(* PLC project Untitled1, Eclipse Foundation CIF to Structured Text 0.0 *)
(* stored: creationDateTime 1970-01-01T00:00:00Z *)

TYPE STATE : STRUCT
  curTime : LREAL;
  dvar_M_aut_i AT %Q* : DINT;
  dvar_M_aut_j AT %Q* : DINT;
  dvar_M_aut_l AT %Q* : ARRAY[0..4] OF DINT;
  dvar_M_aut_ll AT %Q* : ARRAY[0..1] OF ARRAY[0..4] OF DINT;
  dvar_M_aut_empty_arr AT %Q* : ARRAY[0..0] OF DINT;
  dvar_M_aut AT %Q* : enum_E;
END_STRUCT;
END_TYPE

TYPE enum_E : (elit_l1, elit_l2, elit_l3, elit_l4, elit_l5, elit_l6, elit_l7, elit_l8);
END_TYPE

FUNCTION makeArray0 : ARRAY[0..4] OF DINT
  VAR_INPUT
    elem0 : DINT;
    elem1 : DINT;
    elem2 : DINT;
    elem3 : DINT;
    elem4 : DINT;
  END_VAR
  VAR
    rslt : ARRAY[0..4] OF DINT;
  END_VAR

            rslt[0] := elem0;
rslt[1] := elem1;
rslt[2] := elem2;
rslt[3] := elem3;
rslt[4] := elem4;
makeArray0 := rslt;
          
END_FUNCTION

FUNCTION normProjIdx : DINT
  VAR_INPUT
    idx : DINT;
    size : DINT;
  END_VAR
  VAR
    tmp : DINT;
  END_VAR

            tmp := idx;
IF tmp < 0 THEN
    tmp := size + tmp;
END_IF;
normProjIdx := tmp;
          
END_FUNCTION

FUNCTION projArray0 : DINT
  VAR_INPUT
    arr : ARRAY[0..4] OF DINT;
    idx : DINT;
  END_VAR

            projArray0 := arr[normProjIdx(idx, 5)];
          
END_FUNCTION

FUNCTION func_pf : DINT
  VAR_INPUT
    farg_pf_x : DINT;
  END_VAR

            func_pf := projArray0(makeArray0(1, 2, 3, 4, 5), farg_pf_x);
RETURN;
          
END_FUNCTION

FUNCTION func_lf : ARRAY[0..4] OF DINT
  VAR_INPUT
    farg_lf_l : ARRAY[0..4] OF DINT;
    farg_lf_x : DINT;
  END_VAR
  VAR
    fvar_lf_r : ARRAY[0..4] OF DINT;
  END_VAR

            // Initialize local variables.
fvar_lf_r := farg_lf_l;

// Actual function body.
fvar_lf_r[normProjIdx(farg_lf_x, 5)] := 6;
func_lf := fvar_lf_r;
RETURN;
          
END_FUNCTION

FUNCTION makeArray1 : ARRAY[0..1] OF ARRAY[0..4] OF DINT
  VAR_INPUT
    elem0 : ARRAY[0..4] OF DINT;
    elem1 : ARRAY[0..4] OF DINT;
  END_VAR
  VAR
    rslt : ARRAY[0..1] OF ARRAY[0..4] OF DINT;
  END_VAR

            rslt[0] := elem0;
rslt[1] := elem1;
makeArray1 := rslt;
          
END_FUNCTION

FUNCTION func_llf : ARRAY[0..1] OF ARRAY[0..4] OF DINT
  VAR_INPUT
    farg_llf_x : DINT;
    farg_llf_y : DINT;
  END_VAR
  VAR
    fvar_llf_r : ARRAY[0..1] OF ARRAY[0..4] OF DINT;
  END_VAR

            // Initialize local variables.
fvar_llf_r := makeArray1(makeArray0(1, 2, 3, 4, 5), makeArray0(1, 2, 3, 4, 5));

// Actual function body.
fvar_llf_r[normProjIdx(0, 2)][normProjIdx(farg_llf_x, 5)] := farg_llf_y;
func_llf := fvar_llf_r;
RETURN;
          
END_FUNCTION

FUNCTION makeArray2 : ARRAY[0..0] OF DINT
  VAR_INPUT
    elem0 : DINT;
  END_VAR
  VAR
    rslt : ARRAY[0..0] OF DINT;
  END_VAR

            rslt[0] := elem0;
makeArray2 := rslt;
          
END_FUNCTION

FUNCTION projArray1 : ARRAY[0..4] OF DINT
  VAR_INPUT
    arr : ARRAY[0..1] OF ARRAY[0..4] OF DINT;
    idx : DINT;
  END_VAR

            projArray1 := arr[normProjIdx(idx, 2)];
          
END_FUNCTION

PROGRAM MAIN
  VAR_OUTPUT
    timerValue0 : TIME;
    timerValue1 : TIME;
  END_VAR
  VAR
    cnt : LINT;
    first : BOOL := TRUE;
    curTimerValue : TIME;
    state0 : STATE;
    curTime : LREAL;
    loopsKilled : LINT;
  END_VAR
  VAR_TEMP
    lastTimerValue : TIME;
    curDeltaTime : TIME;
    curDeltaSecs : LREAL;
    state1 : STATE;
    progress : BOOL;
    loopCount : INT;
  END_VAR

            
// Handle 'time' and cycle time.
cnt := cnt + 1;

timer0(IN := curTimer = 0, PT := T#1D);
timer1(IN := curTimer = 1, PT := T#1D);
timerValue0 := timer0.ET;
timerValue1 := timer1.ET;

lastTimerValue := curTimerValue;
IF curTimer = 0 THEN
    curTimerValue := timerValue0;
ELSE
    curTimerValue := timerValue1;
END_IF;
curDeltaTime := curTimerValue - lastTimerValue;
curDeltaSecs := TIME_TO_LREAL(curDeltaTime) / 1000;
curTime := curTime + curDeltaSecs;

IF cnt MOD 10 = 0 THEN
    curTimer := 1 - curTimer;
    curTimerValue := T#0S;
    timer0(IN := curTimer = 0, PT := T#1D);
    timer1(IN := curTimer = 1, PT := T#1D);
    timerValue0 := timer0.ET;
    timerValue1 := timer1.ET;
END_IF;

IF first THEN
    first := FALSE;

    // Initialize state variables for initial state.
    state0.dvar_M_aut_i := 0;
    state0.dvar_M_aut_j := 1;
    state0.dvar_M_aut_l := makeArray0(1, 2, 3, 4, 5);
    state0.dvar_M_aut_ll := makeArray1(makeArray0(1, 2, 3, 4, 5), makeArray0(1, 2, 3, 4, 5));
    state0.dvar_M_aut_empty_arr := makeArray2();
    state0.dvar_M_aut := elit_l1;
ELSE
    // Update continuous variables for time delay.

    state0.curTime := curTime;
END_IF;

// Event loop.
WHILE TRUE DO
    progress := FALSE;

    // Event "tau".
    IF NOT progress THEN
        IF (state0.dvar_M_aut) = (elit_l1) THEN
            progress := TRUE;
            state1 := state0;

            state1.dvar_M_aut_i := state0.dvar_M_aut_l[normProjIdx(0, 5)];
            state1.dvar_M_aut_j := state0.dvar_M_aut_l[normProjIdx(-1, 5)];
            state1.dvar_M_aut := elit_l2;

            state0 := state1;
        END_IF;
    END_IF;

    // Event "tau".
    IF NOT progress THEN
        IF (state0.dvar_M_aut) = (elit_l2) THEN
            progress := TRUE;
            state1 := state0;

            state1.dvar_M_aut_l[normProjIdx(0, 5)] := 7;
            state1.dvar_M_aut_l[normProjIdx(-1, 5)] := 8;
            state1.dvar_M_aut := elit_l3;

            state0 := state1;
        END_IF;
    END_IF;

    // Event "tau".
    IF NOT progress THEN
        IF (state0.dvar_M_aut) = (elit_l3) THEN
            progress := TRUE;
            state1 := state0;

            state1.dvar_M_aut_ll[normProjIdx(-2, 2)] := func_lf(makeArray0(11, 22, 33, 44, 55), -1);
            state1.dvar_M_aut := elit_l4;

            state0 := state1;
        END_IF;
    END_IF;

    // Event "tau".
    IF NOT progress THEN
        IF (state0.dvar_M_aut) = (elit_l4) THEN
            progress := TRUE;
            state1 := state0;

            state1.dvar_M_aut_ll := func_llf(-1, 9);
            state1.dvar_M_aut := elit_l5;

            state0 := state1;
        END_IF;
    END_IF;

    // Event "tau".
    IF NOT progress THEN
        IF (state0.dvar_M_aut) = (elit_l5) THEN
            progress := TRUE;
            state1 := state0;

            state1.dvar_M_aut_ll[normProjIdx(0, 2)] := projArray1(func_llf(3, 123), 0);
            state1.dvar_M_aut := elit_l6;

            state0 := state1;
        END_IF;
    END_IF;

    // Event "tau".
    IF NOT progress THEN
        IF (state0.dvar_M_aut) = (elit_l6) THEN
            progress := TRUE;
            state1 := state0;

            state1.dvar_M_aut_i := projArray0(state0.dvar_M_aut_ll[normProjIdx(1, 2)], 2);
            state1.dvar_M_aut := elit_l7;

            state0 := state1;
        END_IF;
    END_IF;

    // Event "tau".
    IF NOT progress THEN
        IF (state0.dvar_M_aut) = (elit_l7) THEN
            progress := TRUE;
            state1 := state0;

            state1.dvar_M_aut_empty_arr := makeArray2();
            state1.dvar_M_aut := elit_l8;

            state0 := state1;
        END_IF;
    END_IF;

    // Done with events?
    IF NOT progress THEN
        EXIT;
    END_IF;

    // Protect against events that are always enabled.
    loopCount := loopCount + 1;
    IF loopCount >= 100 THEN
        loopsKilled := loopsKilled + 1;
        EXIT;
    END_IF;
END_WHILE;
          
END_PROGRAM

CONFIGURATION Untitled1
  RESOURCE Untitled1 ON PLC
    VAR_GLOBAL  (* INPUTS *)
      ivar_i AT %I* : DINT;
    END_VAR
    VAR_GLOBAL  (* TIMERS *)
      timer0 : TON;
      timer1 : TON;
      curTimer : INT := 0;
    END_VAR
    TASK PlcTask(INTERVAL := T#10ms, PRIORITY := 20);
    PROGRAM MAIN WITH PlcTask : MAIN;
  END_RESOURCE
END_CONFIGURATION
